ABB RobotStudio station: test_station.rsstn

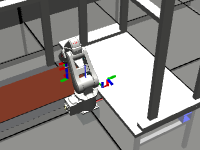
Station Stationstation_server_test (saved by RobotStudio 6.7.7936.1011)
Controller WILL4230
  mechanical unit ROB_1: IRB120_3_58__01, 6 joints, base frame (0, 0, 0) mm
Layout (positions relative to the parent item):
  - IRB120_3_58__01 [mechanism, from Robots\IRB120_3_58_G_01.rslib] at (0, 0, 0) mm; joint values [1.5708, 0.654, 0.2346, 0, 0.6822, 1.5708] (rad or m)
  - Part_1 [part]
  - Part_2 [part]
  - Part_3 [part, from RobotStudio code\WorkArea_Library.rslib]
  - FinalFinalAssembly [part, from RobotStudio code\FinalFinalAssembly_Library.rslib] at (-2915, -5250, -590) mm, rotated rx 180 ry 0 rz 180 deg
  - Block Group [graphiccomponentgroup] at (39, 0, 0) mm
    - Block 1B [part, from Block Libraries\Block 1B.rslib] at (-265, 517, 25) mm
    - Block 1D [part, from Block Libraries\Block 1D.rslib] at (-265, 517, 25) mm
    - Block 1F [part, from Block Libraries\Block 1F.rslib] at (-265, 517, 25) mm
    - Block 1H [part, from Block Libraries\Block 1H.rslib] at (-265, 517, 25) mm
    - Block 3B [part, from Block Libraries\Block 3B.rslib] at (-265, 517, 25) mm
    - Block 3D [part, from Block Libraries\Block 3D.rslib] at (-265, 517, 25) mm
    - Block 3F [part, from Block Libraries\Block 3F.rslib] at (-266, 517, 25) mm
    - Block 3H [part, from Block Libraries\Block 3H.rslib] at (-265, 517, 25) mm
    - Block 5B [part, from Block Libraries\Block 5B.rslib] at (-265, 517, 25) mm
    - Block 5D [part, from Block Libraries\Block 5D.rslib] at (-265, 517, 25) mm
    - Block 5f [part, from Block Libraries\Block 5f.rslib] at (-265, 517, 25) mm
    - Block 5H [part, from Block Libraries\Block 5H.rslib] at (-265, 517, 25) mm
    - Block 7B [part, from Block Libraries\Block 7B.rslib] at (-265, 517, 25) mm
    - Block 7D [part, from Block Libraries\Block 7D.rslib] at (-265, 445, 25) mm
    - Block 7F [part, from Block Libraries\Block 7F.rslib] at (-265, 445, 25) mm
    - Block 7H [part, from Block Libraries\Block 7H.rslib] at (-265, 445, 25) mm
  - Attacher [smart component, from Components\Attacher.rslib]
      properties: Parent=IRB120_3_58__01; Flange=0; Child=Block 1H; Mount=false; Offset=[0 0 0]; Orientation=[0 0 0]
  - Detacher [smart component, from Components\Detacher.rslib]
      properties: Child=Block 1H; KeepPosition=true
  - CollisionSensor [smart component, from Components\CollisionSensor.rslib]
      properties: Object1=SuctionCup; Object2=Block Group; NearMiss=0.01; Part1=SuctionCup; Part2=Block 1H; CollisionType=2
  - SuctionCup [part] at (0, 409, 242) mm, rotated rx -180 ry 0 rz 180 deg
  - wTable [frame] at (175, 0, 147) mm
Attachment: SuctionCup is attached to IRB120_3_58__01 / Link6
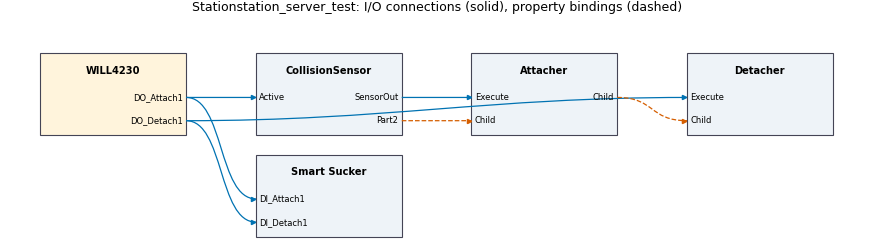
Station logic (signal -> signal, property => property):
  WILL4230.DO_Attach1 -> Smart Sucker.DI_Attach1
  WILL4230.DO_Detach1 -> Smart Sucker.DI_Detach1
  WILL4230.DO_Attach1 -> CollisionSensor.Active
  CollisionSensor.SensorOut -> Attacher.Execute
  WILL4230.DO_Detach1 -> Detacher.Execute
  CollisionSensor.Part2 => Attacher.Child
  Attacher.Child => Detacher.Child
Targets, tools, work objects and paths stored in the station, written as RAPID:
! task T_ROB1
MODULE MTRN_Rob_Data
  PERS wobjdata wTable:=[FALSE,TRUE,"",[[175,0,147],[1,0,0,0]],[[0,0,0],[1,0,0,0]]];
  PERS wobjdata wConveyer:=[FALSE,TRUE,"",[[0,409,22],[0.707106781,0,0,0.707106781]],[[0,0,0],[1,0,0,0]]];
  PERS wobjdata wConveyerCamera:=[FALSE,TRUE,"",[[-71,429,1110],[1,0,0,0]],[[0,0,0],[1,0,0,0]]];
  PERS wobjdata wTableCamera:=[FALSE,TRUE,"",[[309,19,1110],[1,0,0,0]],[[0,0,0],[1,0,0,0]]];
  PERS wobjdata wWorld:=[FALSE,TRUE,"",[[-3025,-3282,-585],[1,0,0,0]],[[0,0,0],[1,0,0,0]]];
  PERS wobjdata wEffector:=[FALSE,TRUE,"",[[0,-374,630],[0.5,0.5,0.5,-0.5]],[[0,0,0],[1,0,0,0]]];
  PERS wobjdata wBase:=[FALSE,TRUE,"",[[0,0,0],[1,0,0,0]],[[0,0,0],[1,0,0,0]]];
  PERS tooldata tSCup:=[TRUE,[[0,0,65],[1,0,0,0]],[0.5,[0,0,20],[1,0,0,0],0,0,0]];
  PERS wobjdata wConv:=[FALSE,TRUE,"",[[50,184,22],[0.5,-0.5,0.5,0.5]],[[1,1,1],[1,0,0,0]]];
  PERS wobjdata Workobject_2:=[FALSE,TRUE,"",[[175,0,147],[1,0,0,0]],[[0,0,0],[1,0,0,0]]];
  CONST jointtarget jtCalibPos:=[[-90,0,0,0,0,0],[9E+09,9E+09,9E+09,9E+09,9E+09,9E+09]];
ENDMODULE

! task T_ROB1
MODULE ROB_MAIN
  PERS wobjdata wobjCurrent:=[FALSE,TRUE,"",[[0,0,0],[1,0,0,0]],[[0,0,0],[1,0,0,0]]];
  PROC Main()
    MoveToCalibPos;
    SingArea \Wrist;
    ConfJ \On;
    MoveToCalibPos;
    vacPwrOff;
    vacSolOff;
    conRunOff;
    conDirRob;
    conRunOn;
    conRunOff;
    conDirHome;
    conDirRob;
    vacSolOn;
    vacSolOff;
    vacPwrOn;
    vacPwrOff;
  ENDPROC
  PROC vacPwrOn()
    SetDO DO10_1,1;
  ENDPROC
  PROC vacPwrOff()
    SetDO DO10_1,0;
  ENDPROC
  PROC vacSolOn()
    SetDO DO10_2,1;
  ENDPROC
  PROC vacSolOff()
    SetDO DO10_2,0;
  ENDPROC
  PROC conRunOn()
    SetDO DO10_3,1;
  ENDPROC
  PROC conRunOff()
    SetDO DO10_3,0;
  ENDPROC
  PROC conDirRob()
    SetDO DO10_4,1;
  ENDPROC
  PROC conDirHome()
    SetDO DO10_4,0;
  ENDPROC
ENDMODULE

! task T_ROB1
MODULE MTRN_Rob_Proc
  PROC MoveToCalibPos()
    MoveAbsJ jtCalibPos,v400,fine,tool0;
  ENDPROC
ENDMODULE

